// TwinCAT 3 PLC project PLC1
// ProgramVersion: 3.1.4024.0
// libraries:
//   Tc2_Math, * (Beckhoff Automation GmbH)
//   Tc2_Standard, * (Beckhoff Automation GmbH)
//   Tc2_System, * (Beckhoff Automation GmbH)
//   Tc3_Module, * (Beckhoff Automation GmbH)
// project tree:
//   / PlcTask.TcTTO
//   Programs/ MAIN.TcPOU
//   RoundLREAL/ fnRoundLREAL.TcPOU, fnRoundLREAL_TRUNC.TcPOU
// real-time tasks:
//   TASK PlcTask: cycle T#10ms, priority 20, ADS port 350

CONFIGURATION PLC1
    RESOURCE PLC ON TwinCAT3
        TASK PlcTask(INTERVAL := T#10ms, PRIORITY := 20);
        PROGRAM MAIN WITH PlcTask : MAIN;
    END_RESOURCE
END_CONFIGURATION

// ---- Programs/MAIN.TcPOU
PROGRAM MAIN
VAR
	RawNumber		:LREAL := 2.56870000002;
	DecimalPlaces	:USINT := 3;
	RoundedNumber1	:LREAL;
	RoundedNumber2	:LREAL;
END_VAR

// Method 1: Uses LINT
RoundedNumber1 := fnRoundLREAL(
	NumberToRound := RawNumber,
	Decimals := DecimalPlaces
);

// Method 2: Uses LTRUNC but requires Tc2_Math library
RoundedNumber2 := fnRoundLREAL_TRUNC(
	NumberToRound := RawNumber,
	Decimals := DecimalPlaces
);

END_PROGRAM

// ---- RoundLREAL/fnRoundLREAL.TcPOU
FUNCTION fnRoundLREAL : LREAL
VAR_INPUT
	NumberToRound		:LREAL;		// Number that needs rounding
	Decimals			:USINT;		// Decimal places wanted
END_VAR
VAR
	rRoundREAL		:LREAL;
	iRoundINT		:LINT;
	rMultiplier		:LREAL;	
END_VAR

// Multiplier = 10^Decimals
rMultiplier := EXPT(10, Decimals);

// Shift decimal x positions to the right 
rRoundREAL := (NumberToRound * rMultiplier) + 0.5;

// Round the number by converting it to an integer (use LINT for large numbers) 
iRoundINT := LREAL_TO_LINT(rRoundREAL);

// Shift decimal x potions back to the left
rRoundREAL := LINT_TO_LREAL(iRoundINT) / rMultiplier;

// Return result
fnRoundLReal := rRoundREAL;

END_FUNCTION

// ---- RoundLREAL/fnRoundLREAL_TRUNC.TcPOU
FUNCTION fnRoundLREAL_TRUNC : LREAL
VAR_INPUT
	NumberToRound		:LREAL;		// Number that needs rounding
	Decimals			:USINT;		// Decimal places wanted
END_VAR
VAR
	rRoundREAL		:LREAL;
	rMultiplier		:LREAL;	
END_VAR

// Multiplier = 10^Decimals
rMultiplier := EXPT(10, Decimals);

// Shift decimal x positions to the right 
rRoundREAL := (NumberToRound * rMultiplier) + 0.5;

// Round the number by converting it to an integer (use LINT for large numbers) 
rRoundREAL := LTRUNC(rRoundREAL);

// Shift decimal x potions back to the left
rRoundREAL := rRoundREAL / rMultiplier;

// Return result
fnRoundLREAL_TRUNC := rRoundREAL;

END_FUNCTION
